// TIA Portal V17 export
ORGANIZATION_BLOCK "Main"   // OB1, SCL, ProgramCycle
   VAR_INPUT
      Initial_Call : Bool;
      Remanence : Bool;
   END_VAR
   VAR_TEMP
      speed : Real;
   END_VAR
BEGIN
   "Conveyor_DB"(Start := "Start_Button", Stop := "Stop_Button");
   // vitesse en tr/min
   #speed := INT_TO_REAL(in := "Conveyor_DB".Count) * 2.5;
   IF %M10.1 THEN
       "Speed_Display" := #speed;
   END_IF;
END_ORGANIZATION_BLOCK
